// TIA Portal project "kazan_suyu_sicakliği" (V18)

(* hardware
DEVICE "S7-1200 station_1"  S7-1200 Station
   slot 0: "Rack_0"  S7-1200 Rack  Rack  V1.0
   slot 1: "PLC_1"  CPU 1214C DC/DC/DC  6ES7 214-1AG40-0XB0  V4.6
*)

// ===== PLC "PLC_1"  CPU 1214C DC/DC/DC =====

VAR_GLOBAL   // PLC tag table "Default tag table"
   "Tag_1" AT %IW64 : Int;
   "Tag_2" AT %MD0 : Real;
   "Tag_3" AT %Q0.0 : Bool;
END_VAR

DATA_BLOCK "iki_nokta_kontrollü_uygulama_DB"   // DB1
{ S7_Optimized_Access := 'TRUE' }
VERSION : 0.1
// stored: InstanceOfName iki_nokta_kontrollü_uygulama
"iki_nokta_kontrollü_uygulama"
BEGIN
END_DATA_BLOCK

FUNCTION_BLOCK "iki_nokta_kontrollü_uygulama"   // FB1, LAD
{ S7_Optimized_Access := 'TRUE' }
VERSION : 0.1
   VAR_INPUT
      "SET DEĞERİ" : Int;
      "GERÇEK DEĞER" : Int;
      "HATA ORANI" : Real;
   END_VAR
   VAR_OUTPUT
      ISITICI : Bool;
   END_VAR
   VAR_IN_OUT
      SICAKLIK : Real;
   END_VAR
   VAR
      "ALT SINIR" : Real;
      "ÜST SINIR" : Real;
      "ANAHTARLAMA ARALIĞI" : Real;
      "SET REAL" : Real;
      "GERÇEK DEĞER REAL" : Real;
   END_VAR
BEGIN

REGION Network 1
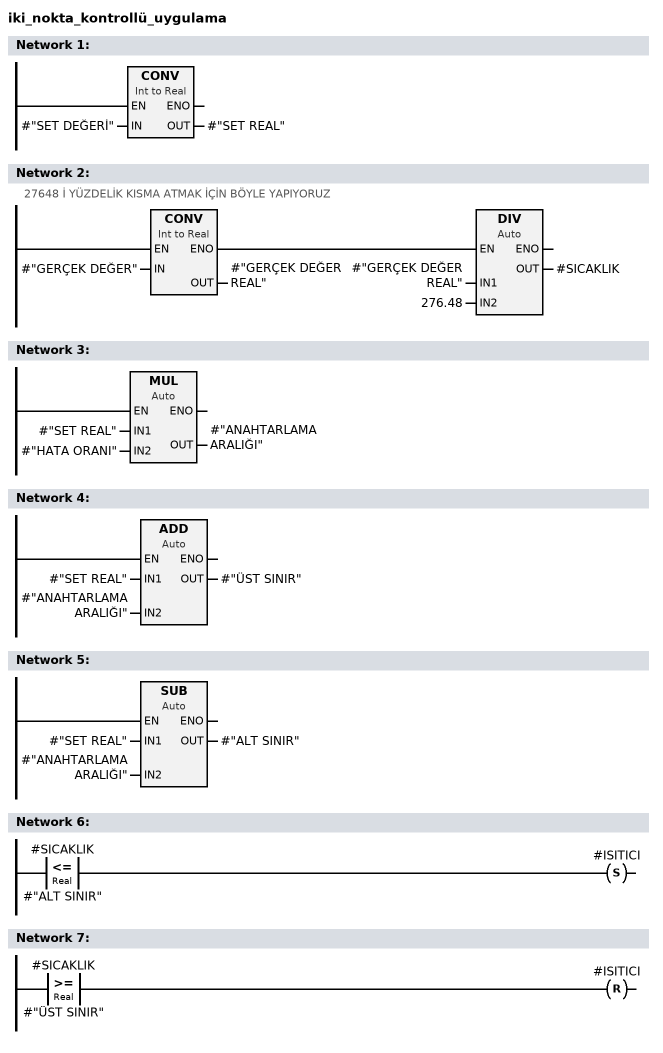
   RUNG wire#powerrail
      { S7_Templates := "[SrcType := Int, DestType := Real]" } Convert(in := #"SET DEĞERİ", out => #"SET REAL")
   END_RUNG
   // the same network as SCL:
   #"SET REAL" := INT_TO_REAL(#"SET DEĞERİ");
END_REGION

REGION Network 2
   // 27648 İ YÜZDELİK KISMA ATMAK İÇİN BÖYLE YAPIYORUZ
   RUNG wire#powerrail
      { S7_Templates := "[SrcType := Int, DestType := Real]" } Convert(in := #"GERÇEK DEĞER", out => #"GERÇEK DEĞER REAL")
      Div(in1 := #"GERÇEK DEĞER REAL", in2 := 276.48, out => #SICAKLIK)
   END_RUNG
   // the same network as SCL:
   #"GERÇEK DEĞER REAL" := INT_TO_REAL(#"GERÇEK DEĞER");
   #SICAKLIK := #"GERÇEK DEĞER REAL" / 276.48;
END_REGION

REGION Network 3
   RUNG wire#powerrail
      Mul(in1 := #"SET REAL", in2 := #"HATA ORANI", out => #"ANAHTARLAMA ARALIĞI")
   END_RUNG
   // the same network as SCL:
   #"ANAHTARLAMA ARALIĞI" := #"SET REAL" * #"HATA ORANI";
END_REGION

REGION Network 4
   RUNG wire#powerrail
      Add(in1 := #"SET REAL", in2 := #"ANAHTARLAMA ARALIĞI", out => #"ÜST SINIR")
   END_RUNG
   // the same network as SCL:
   #"ÜST SINIR" := #"SET REAL" + #"ANAHTARLAMA ARALIĞI";
END_REGION

REGION Network 5
   RUNG wire#powerrail
      Sub(in1 := #"SET REAL", in2 := #"ANAHTARLAMA ARALIĞI", out => #"ALT SINIR")
   END_RUNG
   // the same network as SCL:
   #"ALT SINIR" := #"SET REAL" - #"ANAHTARLAMA ARALIĞI";
END_REGION

REGION Network 6
   RUNG wire#powerrail
      { S7_Templates := "SrcType := Real" } LE_Contact(in1 := #SICAKLIK, in2 := #"ALT SINIR")
      S_Coil( #ISITICI )
   END_RUNG
   // the same network as SCL:
   IF #SICAKLIK <= #"ALT SINIR" THEN #ISITICI := TRUE; END_IF;
END_REGION

REGION Network 7
   RUNG wire#powerrail
      { S7_Templates := "SrcType := Real" } GE_Contact(in1 := #SICAKLIK, in2 := #"ÜST SINIR")
      R_Coil( #ISITICI )
   END_RUNG
   // the same network as SCL:
   IF #SICAKLIK >= #"ÜST SINIR" THEN #ISITICI := FALSE; END_IF;
END_REGION
END_FUNCTION_BLOCK

ORGANIZATION_BLOCK "Main"   // OB1, LAD, ProgramCycle
TITLE = "Main Program Sweep (Cycle)"
{ S7_Optimized_Access := 'TRUE' }
VERSION : 0.1
   VAR_INPUT
      Initial_Call : Bool;   // Initial call of this OB
      Remanence : Bool;   // =True, if remanent data are available
   END_VAR
BEGIN

REGION Network 1
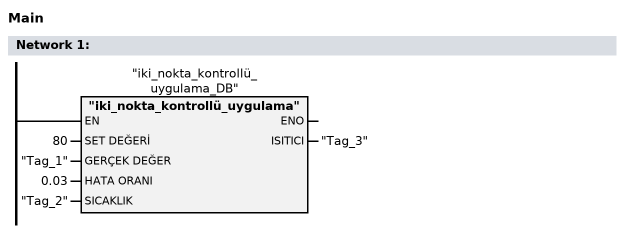
   RUNG wire#powerrail
      "iki_nokta_kontrollü_uygulama_DB"("SET DEĞERİ" := 80, "GERÇEK DEĞER" := "Tag_1", "HATA ORANI" := 0.03, SICAKLIK := "Tag_2", ISITICI => "Tag_3")
   END_RUNG
   // the same network as SCL:
   "iki_nokta_kontrollü_uygulama_DB"("SET DEĞERİ" := 80,   // "iki_nokta_kontrollü_uygulama"
                           "GERÇEK DEĞER" := "Tag_1",
                           "HATA ORANI" := 0.03,
                           SICAKLIK := "Tag_2",
                           ISITICI => "Tag_3");
END_REGION
END_ORGANIZATION_BLOCK